FUNCTION_BLOCK PUBL_8_SETUP (* 8-variable local group publisher for setup resource *)
  (* Standard: 61499-2 *)
  (* Version 1.0, 13-04-12, GASR, Universidade do Estado de Santa Catarina *)
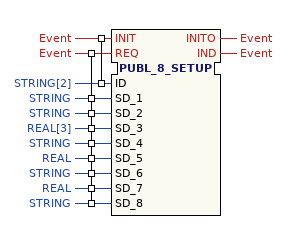
  EVENT_INPUT
    INIT WITH ID; (* Service Initialization *)
    REQ WITH SD_1, SD_2, SD_3, SD_4, SD_5, SD_6, SD_7, SD_8; (* Service Request *)
  END_EVENT
  EVENT_OUTPUT
    INITO; (* Initialization Confirm *)
    IND; (* Service Confirmation *)
  END_EVENT
  VAR_INPUT
    ID : ARRAY [0..1] OF STRING; (* Default id is the FB instance name *)
    SD_1 : STRING; (* workplan.its_setup.its_origin.name *)
    SD_2 : STRING; (* workplan.its_setup.its_origin.location.name *)
    SD_3 : ARRAY [0..2] OF REAL; (* workplan.its_setup.its_origin.location.coordinates *)
    SD_4 : STRING; (* workplan.its_setup.its_origin.axis.its_id *)
    SD_5 : REAL; (* workplan.its_setup.its_origin.axis.direction_ratios *)
    SD_6 : STRING; (* workplan.its_setup.its_origin.ref_direction.its_id *)
    SD_7 : REAL; (* workplan.its_setup.its_origin.ref_direction_ratios *)
    SD_8 : STRING; (* current_tool *)
  END_VAR
  SERVICE PUBL_8_SETUP/SUBL_8_SETUP (* Data publication service *)
    SEQUENCE normal_establishment
      PUBL_8_SETUP.INIT(ID) -> PUBL_8_SETUP.INITO();
      SUBL_8_SETUP.INIT(ID) -> SUBL_8_SETUP.INITO();
    END_SEQUENCE
    SEQUENCE normal_data_transfer
      PUBL_8_SETUP.REQ(SD_1,SD_2,SD_3,SD_4,SD_5,SD_6,SD_7,SD_8) -> SUBL_8_SETUP.IND(RD_1,RD_2,RD_3,RD_4,RD_5,RD_6,RD_7,RD_8) -> PUBL_8_SETUP.CNF();
    END_SEQUENCE
  END_SERVICE
END_FUNCTION_BLOCK
